Fanuc KAREL source: kt00974.KL

PROGRAM KT00974
%STACKSIZE=65535
%PRIORITY=65535
%NOLOCKGROUP
VAR
ENTRY : INTEGER
PNAME : STRING[80]
VNAME : STRING[80]
STATUS : INTEGER
-- UNRESOLVED DECLARATIONS (source type spelling not recovered)
-- VALUE : ARRAY[4] OF TYPE_0x0013 (type_u16=0x2013)
BEGIN
ENTRY=0
PNAME=''
VNAME='VALUE'
-- UNRESOLVED_PC line 13 opcodes [27 22 22 2A 22 2A 22 22 B0] marker_code=43
END KT00974
